// Mitsubishi GX Developer project: PLC_PCO520L2   PLC: Q06UDEH

PROGRAM RECIPE
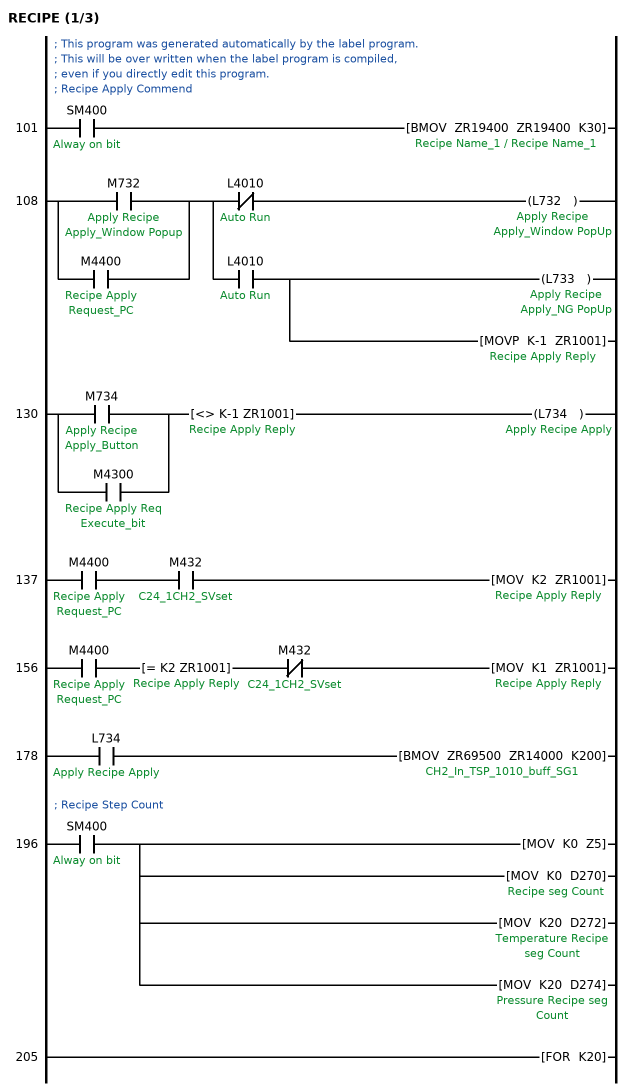
; This program was generated automatically by the label program.
; This will be over written when the label program is compiled,
; even if you directly edit this program.
; Recipe Apply Commend
101   LD      SM400  ; Alway on bit
      BMOV    ZR19400 ZR19400 K30  ; Recipe Name_1
108   LD      M732  ; Apply Recipe Apply_Window Popup
      OR      M4400  ; Recipe Apply Request_PC
      MPS
      ANI     L4010  ; Auto Run
      OUT     L732  ; Apply Recipe Apply_Window PopUp
      MPP
      AND     L4010  ; Auto Run
      OUT     L733  ; Apply Recipe Apply_NG PopUp
      MOVP    K-1 ZR1001  ; Recipe Apply Reply
        [note] Recipe Apply Fail
130   LD      M734  ; Apply Recipe Apply_Button
      OR      M4300  ; Recipe Apply Req Execute_bit
      AND<>   K-1 ZR1001  ; Recipe Apply Reply
      OUT     L734  ; Apply Recipe Apply
137   LD      M4400  ; Recipe Apply Request_PC
      AND     M432  ; C24_1CH2_SVset
      MOV     K2 ZR1001
        [note] Recipe apply inprogress
156   LD      M4400  ; Recipe Apply Request_PC
      AND=    K2 ZR1001  ; Recipe Apply Reply
      ANI     M432  ; C24_1CH2_SVset
      MOV     K1 ZR1001
        [note] Recipe apply complete
178   LD      L734  ; Apply Recipe Apply
      BMOV    ZR69500 ZR14000 K200  ; CH2_In_TSP_1010_buff_SG1
; Recipe Step Count
196   LD      SM400  ; Alway on bit
      MOV     K0 Z5
      MOV     K0 D270  ; Recipe seg Count
      MOV     K20 D272  ; Temperature Recipe seg Count
      MOV     K20 D274  ; Pressure Recipe seg Count
205   FOR     K20
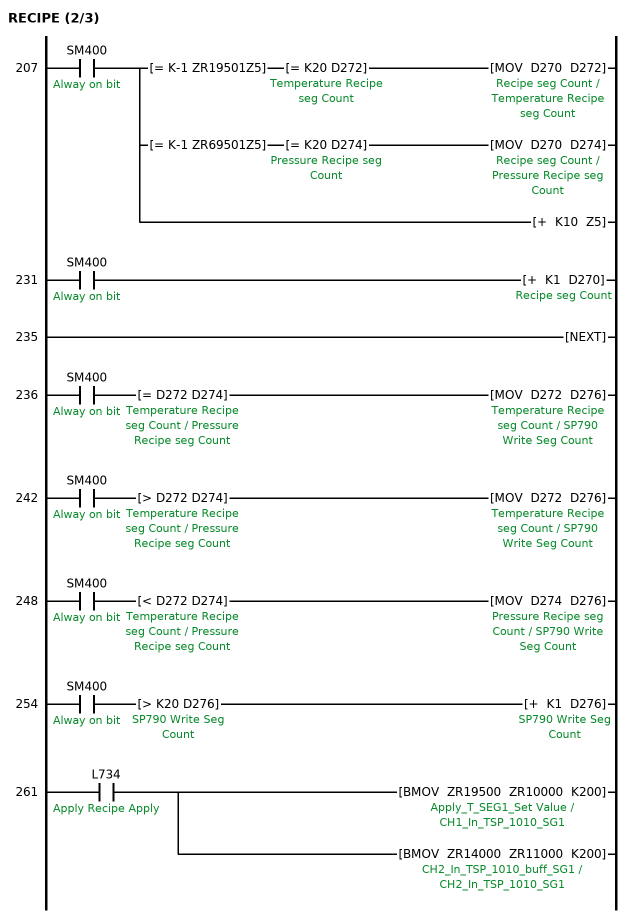
207   LD      SM400  ; Alway on bit
      MPS
      AND=    K-1 ZR19501Z5
      AND=    K20 D272  ; Temperature Recipe seg Count
      MOV     D270 D272
      MRD
      AND=    K-1 ZR69501Z5
      AND=    K20 D274  ; Pressure Recipe seg Count
      MOV     D270 D274
      MPP
      +       K10 Z5
231   LD      SM400  ; Alway on bit
      +       K1 D270
235   NEXT
236   LD      SM400  ; Alway on bit
      AND=    D272 D274  ; Temperature Recipe seg Count / Pressure Recipe seg Count
      MOV     D272 D276  ; SP790 Write Seg Count
242   LD      SM400  ; Alway on bit
      AND>    D272 D274  ; Temperature Recipe seg Count / Pressure Recipe seg Count
      MOV     D272 D276
248   LD      SM400  ; Alway on bit
      AND<    D272 D274  ; Temperature Recipe seg Count / Pressure Recipe seg Count
      MOV     D274 D276
254   LD      SM400  ; Alway on bit
      AND>    K20 D276  ; SP790 Write Seg Count
      +       K1 D276
261   LD      L734  ; Apply Recipe Apply
      BMOV    ZR19500 ZR10000 K200  ; Apply_T_SEG1_Set Value / CH1_In_TSP_1010_SG1
      BMOV    ZR14000 ZR11000 K200  ; CH2_In_TSP_1010_SG1
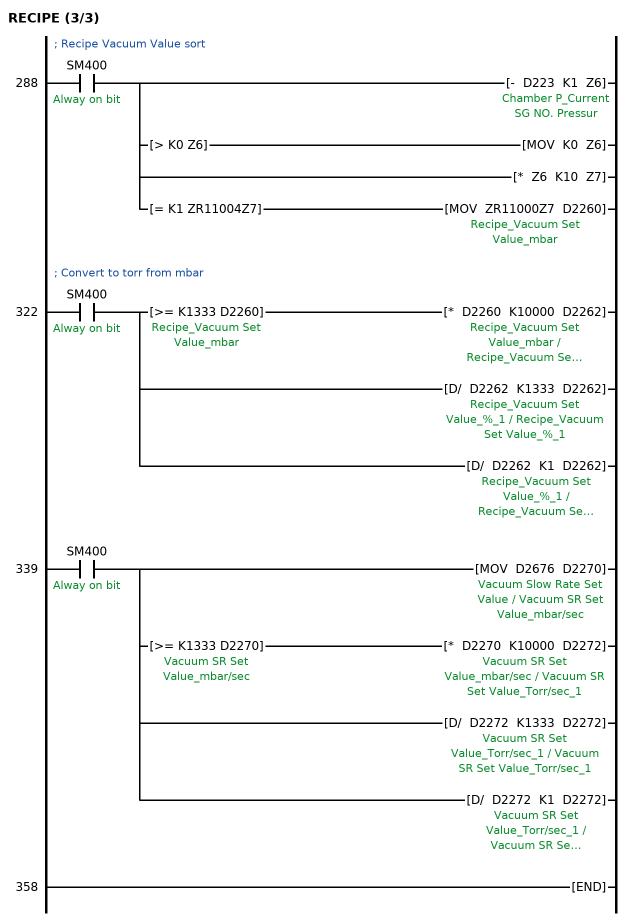
; Recipe Vacuum Value sort
288   LD      SM400  ; Alway on bit
      -       D223 K1 Z6  ; Chamber P_Current SG NO. Pressur
      MPS
      AND>    K0 Z6
      MOV     K0 Z6
      MPP
      *       Z6 K10 Z7
      AND=    K1 ZR11004Z7
      MOV     ZR11000Z7 D2260  ; Recipe_Vacuum Set Value_mbar
; Convert to torr from mbar
322   LD      SM400  ; Alway on bit
      MPS
      AND>=   K1333 D2260  ; Recipe_Vacuum Set Value_mbar
      *       D2260 K10000 D2262  ; Recipe_Vacuum Set Value_%_1
      MPP
      D/      D2262 K1333 D2262
      D/      D2262 K1 D2262
339   LD      SM400  ; Alway on bit
      MOV     D2676 D2270  ; Vacuum Slow Rate Set Value / Vacuum SR Set Value_mbar/sec
      MPS
      AND>=   K1333 D2270  ; Vacuum SR Set Value_mbar/sec
      *       D2270 K10000 D2272  ; Vacuum SR Set Value_Torr/sec_1
      MPP
      D/      D2272 K1333 D2272
      D/      D2272 K1 D2272
358   END
END_PROGRAM
